Fanuc KAREL source: KT00655.KL

PROGRAM KT00655
%NOLOCKGROUP
VAR
  P1: POSITION
  P2: POSITION
  OUT: INTEGER
BEGIN
  OUT = + P1
END KT00655
